REGION Network 135: READ-IN DISABLE
   RUNG wire#powerrail
      I_Contact( "DB362_M_UNIT_02_STA_3".M_CODES_UNIT_02_STA_3.M27 )
      I_Contact( "DB362_M_UNIT_02_STA_3".M_CODES_UNIT_02_STA_3.M28 )
      I_Contact( "DB362_M_UNIT_02_STA_3".M_CODES_UNIT_02_STA_3.M60 )
      I_Contact( "DB362_M_UNIT_02_STA_3".M_CODES_UNIT_02_STA_3.M61 )
      I_Contact( "DB362_M_UNIT_02_STA_3".M_CODES_UNIT_02_STA_3.M100 )
      I_Contact( "DB362_M_UNIT_02_STA_3".M_CODES_UNIT_02_STA_3.M101 )
      I_Contact( "DB362_M_UNIT_02_STA_3".M_CODES_UNIT_02_STA_3.M102 )
      I_Contact( "DB362_M_UNIT_02_STA_3".M_CODES_UNIT_02_STA_3.M103 )
      I_Contact( "DB362_M_UNIT_02_STA_3".M_CODES_UNIT_02_STA_3.M130 )
      I_Contact( "DB362_M_UNIT_02_STA_3".M_CODES_UNIT_02_STA_3.M131 )
      I_Contact( "DB362_M_UNIT_02_STA_3".M_CODES_UNIT_02_STA_3.M150 )
      I_Contact( "DB362_M_UNIT_02_STA_3".M_CODES_UNIT_02_STA_3.M151 )
      I_Contact( "DB362_M_UNIT_02_STA_3".M_CODES_UNIT_02_STA_3.M154 )
      I_Contact( "DB362_M_UNIT_02_STA_3".M_CODES_UNIT_02_STA_3.M155 )
      I_Contact( "DB362_M_UNIT_02_STA_3".M_CODES_UNIT_02_STA_3.M156 )
      I_Contact( "DB362_M_UNIT_02_STA_3".M_CODES_UNIT_02_STA_3.M157 )
      I_Contact( "DB362_M_UNIT_02_STA_3".M_CODES_UNIT_02_STA_3.M164 )
      Not()
      Coil( "DB362_M_UNIT_02_STA_3".M_CODES_UNIT_02_STA_3.READ_IN_DISABLE_GENERAL )
   END_RUNG
   // the same network as SCL:
   "DB362_M_UNIT_02_STA_3".M_CODES_UNIT_02_STA_3.READ_IN_DISABLE_GENERAL := NOT (NOT "DB362_M_UNIT_02_STA_3".M_CODES_UNIT_02_STA_3.M27 AND NOT "DB362_M_UNIT_02_STA_3".M_CODES_UNIT_02_STA_3.M28 AND NOT "DB362_M_UNIT_02_STA_3".M_CODES_UNIT_02_STA_3.M60 AND NOT "DB362_M_UNIT_02_STA_3".M_CODES_UNIT_02_STA_3.M61 AND NOT "DB362_M_UNIT_02_STA_3".M_CODES_UNIT_02_STA_3.M100 AND NOT "DB362_M_UNIT_02_STA_3".M_CODES_UNIT_02_STA_3.M101 AND NOT "DB362_M_UNIT_02_STA_3".M_CODES_UNIT_02_STA_3.M102 AND NOT "DB362_M_UNIT_02_STA_3".M_CODES_UNIT_02_STA_3.M103 AND NOT "DB362_M_UNIT_02_STA_3".M_CODES_UNIT_02_STA_3.M130 AND NOT "DB362_M_UNIT_02_STA_3".M_CODES_UNIT_02_STA_3.M131 AND NOT "DB362_M_UNIT_02_STA_3".M_CODES_UNIT_02_STA_3.M150 AND NOT "DB362_M_UNIT_02_STA_3".M_CODES_UNIT_02_STA_3.M151 AND NOT "DB362_M_UNIT_02_STA_3".M_CODES_UNIT_02_STA_3.M154 AND NOT "DB362_M_UNIT_02_STA_3".M_CODES_UNIT_02_STA_3.M155 AND NOT "DB362_M_UNIT_02_STA_3".M_CODES_UNIT_02_STA_3.M156 AND NOT "DB362_M_UNIT_02_STA_3".M_CODES_UNIT_02_STA_3.M157 AND NOT "DB362_M_UNIT_02_STA_3".M_CODES_UNIT_02_STA_3.M164);
END_REGION
END_FUNCTION
